PROGRAM MAIN
VAR
	text : STRING[30] := 'hello';
END_VAR

END_PROGRAM

(* stored: Version 1.1.0.1, ProductVersion 3.1.4022.3
   POU MAIN: Id {08a38933-7d15-4d08-a1e8-48039f2428b0}, SpecialFunc None *)
